{attribute 'qualified_only'}
VAR_GLOBAL CONSTANT
    // Max direct children a single node may register.
    // Bumped only if a real machine node grows very wide.
    cMaxChildren : DINT := 16;
END_VAR

(* stored: Version 1.1.0.1
   GVL GVL_Framework: Id {bbb6d9da-0c12-4cd1-ae19-153d72597a5a} *)
